# EPICS autosave request: ADApp/Db/NDROIStat_settings.req
# This works for one ROI
$(P)$(R)Name
$(P)$(R)NDArrayCallbacks
$(P)$(R)ROI$(ADDR):Use
$(P)$(R)ROI$(ADDR):MinX
$(P)$(R)ROI$(ADDR):MinY
$(P)$(R)ROI$(ADDR):MinZ
$(P)$(R)ROI$(ADDR):SizeX
$(P)$(R)ROI$(ADDR):SizeY
$(P)$(R)ROI$(ADDR):SizeZ
